FUNCTION_BLOCK SCREW_STATION_MANAGER_NO_SIGNAL
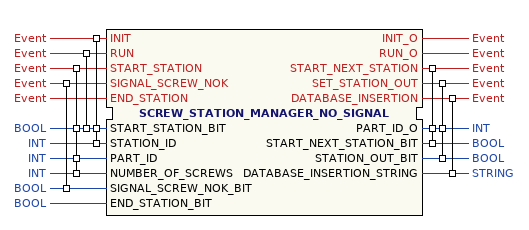
  EVENT_INPUT
    INIT WITH STATION_ID, START_STATION_BIT;
    RUN WITH START_STATION_BIT;
    START_STATION WITH START_STATION_BIT, PART_ID, NUMBER_OF_SCREWS;
    SIGNAL_SCREW_NOK WITH SIGNAL_SCREW_NOK_BIT;
    END_STATION;
  END_EVENT
  EVENT_OUTPUT
    INIT_O;
    RUN_O;
    START_NEXT_STATION WITH PART_ID_O, START_NEXT_STATION_BIT;
    SET_STATION_OUT WITH STATION_OUT_BIT, PART_ID_O;
    DATABASE_INSERTION WITH DATABASE_INSERTION_STRING;
  END_EVENT
  VAR_INPUT
    START_STATION_BIT : BOOL;
    STATION_ID : INT;
    PART_ID : INT;
    NUMBER_OF_SCREWS : INT;
    SIGNAL_SCREW_NOK_BIT : BOOL;
    END_STATION_BIT : BOOL;
  END_VAR
  VAR_OUTPUT
    PART_ID_O : INT;
    START_NEXT_STATION_BIT : BOOL;
    STATION_OUT_BIT : BOOL;
    DATABASE_INSERTION_STRING : STRING;
  END_VAR
END_FUNCTION_BLOCK
